{attribute 'GeneratedUsingTerminal: IODEVICETYPE_ETHERCATPROT'}
{attribute addProperty BoxType "IODEVICETYPE_ETHERCATPROT"}
{attribute addProperty Id "Term_1_EK1100Term_1_EK1100_C62D072D20SyncUnitsSyncUnits_99E584AF18InputsInputs_A65FACA410OutputsOutputs_23C0ED1D6InfoDataInfoData_E68C61CD28"}
{attribute addProperty CRC "2666435239"}
{attribute addProperty Size "82"}
TYPE Device_1_EtherCAT_9EEE92A7 :
STRUCT
	{attribute addProperty Name "Term_1_EK1100"}
	{attribute addProperty PreviousPort "Device 1 (EtherCAT) : Master"}
	Term_1_EK1100 : Term_1_EK1100_C62D072D;
	{attribute addProperty Name "SyncUnits"}
	SyncUnits : SyncUnits_99E584AF;
	{attribute addProperty Name "Inputs"}
	Inputs : TcoIo.Inputs_A65FACA4;
	{attribute addProperty Name "Outputs"}
	Outputs : TcoIo.Outputs_23C0ED1D;
	{attribute addProperty Name "InfoData"}
	InfoData : TcoIo.InfoData_E68C61CD;
END_STRUCT
END_TYPE

(* stored: Version 1.2.0.0, ProductVersion 3.1.4024.9
   DUT Device_1_EtherCAT_9EEE92A7: Id {4fb6f2ff-4285-4355-a37f-43f1c9e5cbd3} *)
